// TIA Portal project "3motorfucnblock" (V20)

(* hardware
DEVICE "S7-1200 station_1"  S7-1200 Station
   slot 0: "Rack_0"  S7-1200 Rack  Rack  V1.0
   slot 1: "PLC_1"  CPU 1214C DC/DC/Rly  6ES7 214-1HG40-0XB0  V4.7
*)

// ===== PLC "PLC_1"  CPU 1214C DC/DC/Rly =====

VAR_GLOBAL   // PLC tag table "Default tag table"
   "Start but 1" AT %I0.0 : Bool;
   "Start but 2" AT %I0.1 : Bool;
   "Start but 3" AT %I0.2 : Bool;
   "Stop but 1" AT %I0.3 : Bool;
   "Stop but 2" AT %I0.4 : Bool;
   "Stop but 3" AT %I0.5 : Bool;
   "Reset but 1" AT %I0.6 : Bool;
   "Reset but 2" AT %I0.7 : Bool;
   "Reset but 3" AT %I1.0 : Bool;
   "Motor 1 çalış" AT %Q0.0 : Bool;
   "Motor 2 çalış" AT %Q0.1 : Bool;
   "Motor 3 çalış" AT %Q0.2 : Bool;
END_VAR

DATA_BLOCK "çalışma zamanları"   // DB1
{ S7_Optimized_Access := 'TRUE' }
VERSION : 0.1
   VAR
      "Motor 1 zaman" : Time := T#5s;
      "Motor 2 zaman" : Time := T#10s;
      "Motor 3 zaman" : Time := T#15s;
   END_VAR
BEGIN
END_DATA_BLOCK

DATA_BLOCK "çalışma sayıları"   // DB2
{ S7_Optimized_Access := 'TRUE' }
VERSION : 0.1
   VAR
      "Motor 1 sayı" : Int := 2;
      "Motor 2 sayı" : Int := 3;
      "Motor 3 sayı" : Int := 4;
   END_VAR
BEGIN
END_DATA_BLOCK

DATA_BLOCK "motor1"   // DB3
{ S7_Optimized_Access := 'TRUE' }
VERSION : 0.1
// stored: InstanceOfName Motorlar
"Motorlar"
BEGIN
END_DATA_BLOCK

DATA_BLOCK "motor2"   // DB4
{ S7_Optimized_Access := 'TRUE' }
VERSION : 0.1
// stored: InstanceOfName Motorlar
"Motorlar"
BEGIN
END_DATA_BLOCK

DATA_BLOCK "motor3"   // DB5
{ S7_Optimized_Access := 'TRUE' }
VERSION : 0.1
// stored: InstanceOfName Motorlar
"Motorlar"
BEGIN
END_DATA_BLOCK

FUNCTION_BLOCK "Motorlar"   // FB1, LAD
{ S7_Optimized_Access := 'TRUE' }
VERSION : 0.1
   VAR_INPUT
      Başlat : Bool;
      Durdur : Bool;
      Resetle : Bool;
      "Çalışma zamanı" : Time;
      "Çalışma sayısı" : Int;
   END_VAR
   VAR_OUTPUT
      "Motor çıkışı" : Bool;
   END_VAR
   VAR
      "Motor hafıza" : Bool;
      timer1 : TON_TIME;
      "Kenar darbesi" : Bool;
      "sayma sonucu" : Int;
      "Yeterli çalışma" : Bool;
   END_VAR
   VAR_TEMP   // added for the SCL form of the ladder/FBD networks
      _w1 : Bool;
   END_VAR
BEGIN

REGION Network 1
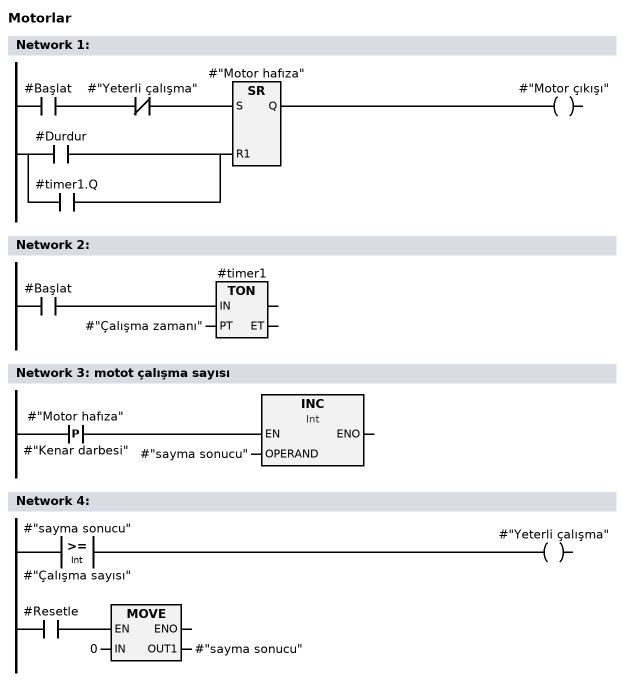
   RUNG wire#powerrail
      Contact( #Başlat )
      I_Contact( #"Yeterli çalışma" )
      S_SR(operand := #"Motor hafıza", r1 := wire#w1)
      Coil( #"Motor çıkışı" )
   END_RUNG
   RUNG wire#powerrail
      Contact( #Durdur )
   END_RUNG wire#w1
   RUNG wire#powerrail
      Contact( #timer1.Q )
   END_RUNG wire#w1
   // the same network as SCL:
   IF #Başlat AND NOT #"Yeterli çalışma" THEN
       #"Motor hafıza" := TRUE;   // SR flip-flop
   END_IF;
   IF #Durdur OR #timer1.Q THEN #"Motor hafıza" := FALSE; END_IF;
   #"Motor çıkışı" := #"Motor hafıza";
END_REGION

REGION Network 2
   #timer1(IN := #Başlat, PT := #"Çalışma zamanı");   // TON
END_REGION

REGION Network 3: motot çalışma sayısı
   RUNG wire#powerrail
      P_Contact(operand := #"Motor hafıza", bit := #"Kenar darbesi")
      { S7_Templates := "DestType := Int" } Inc( #"sayma sonucu" )
   END_RUNG
   // the same network as SCL:
   #_w1 := #"Motor hafıza" AND NOT #"Kenar darbesi";   // rising edge of #"Motor hafıza"
   #"Kenar darbesi" := #"Motor hafıza";
   IF #_w1 THEN #"sayma sonucu" := #"sayma sonucu" + 1; END_IF;
END_REGION

REGION Network 4
   RUNG wire#powerrail
      { S7_Templates := "SrcType := Int" } GE_Contact(in1 := #"sayma sonucu", in2 := #"Çalışma sayısı")
      Coil( #"Yeterli çalışma" )
   END_RUNG
   RUNG wire#powerrail
      Contact( #Resetle )
      Move(in := 0, out1 => #"sayma sonucu")
   END_RUNG
   // the same network as SCL:
   #"Yeterli çalışma" := #"sayma sonucu" >= #"Çalışma sayısı";
   IF #Resetle THEN #"sayma sonucu" := 0; END_IF;
END_REGION
END_FUNCTION_BLOCK

ORGANIZATION_BLOCK "Main"   // OB1, LAD, ProgramCycle
TITLE = "Main Program Sweep (Cycle)"
{ S7_Optimized_Access := 'TRUE' }
VERSION : 0.1
   VAR_INPUT
      Initial_Call : Bool;   // Initial call of this OB
      Remanence : Bool;   // =True, if remanent data are available
   END_VAR
BEGIN

REGION Network 1: Motor 1 çalışma programı
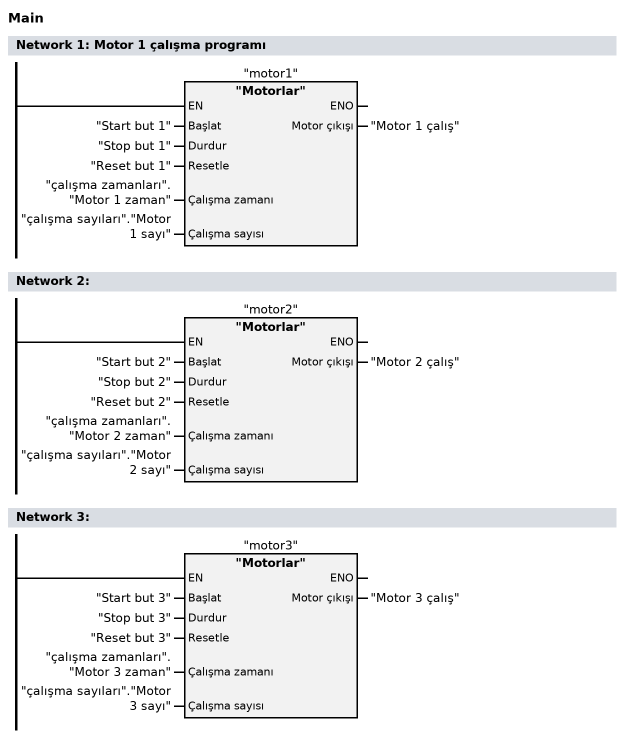
   RUNG wire#powerrail
      "motor1"(Başlat := "Start but 1", Durdur := "Stop but 1", Resetle := "Reset but 1", "Çalışma zamanı" := "çalışma zamanları"."Motor 1 zaman", "Çalışma sayısı" := "çalışma sayıları"."Motor 1 sayı", "Motor çıkışı" => "Motor 1 çalış")
   END_RUNG
   // the same network as SCL:
   "motor1"(Başlat := "Start but 1",   // "Motorlar"
            Durdur := "Stop but 1",
            Resetle := "Reset but 1",
            "Çalışma zamanı" := "çalışma zamanları"."Motor 1 zaman",
            "Çalışma sayısı" := "çalışma sayıları"."Motor 1 sayı",
            "Motor çıkışı" => "Motor 1 çalış");
END_REGION

REGION Network 2
   RUNG wire#powerrail
      "motor2"(Başlat := "Start but 2", Durdur := "Stop but 2", Resetle := "Reset but 2", "Çalışma zamanı" := "çalışma zamanları"."Motor 2 zaman", "Çalışma sayısı" := "çalışma sayıları"."Motor 2 sayı", "Motor çıkışı" => "Motor 2 çalış")
   END_RUNG
   // the same network as SCL:
   "motor2"(Başlat := "Start but 2",   // "Motorlar"
            Durdur := "Stop but 2",
            Resetle := "Reset but 2",
            "Çalışma zamanı" := "çalışma zamanları"."Motor 2 zaman",
            "Çalışma sayısı" := "çalışma sayıları"."Motor 2 sayı",
            "Motor çıkışı" => "Motor 2 çalış");
END_REGION

REGION Network 3
   RUNG wire#powerrail
      "motor3"(Başlat := "Start but 3", Durdur := "Stop but 3", Resetle := "Reset but 3", "Çalışma zamanı" := "çalışma zamanları"."Motor 3 zaman", "Çalışma sayısı" := "çalışma sayıları"."Motor 3 sayı", "Motor çıkışı" => "Motor 3 çalış")
   END_RUNG
   // the same network as SCL:
   "motor3"(Başlat := "Start but 3",   // "Motorlar"
            Durdur := "Stop but 3",
            Resetle := "Reset but 3",
            "Çalışma zamanı" := "çalışma zamanları"."Motor 3 zaman",
            "Çalışma sayısı" := "çalışma sayıları"."Motor 3 sayı",
            "Motor çıkışı" => "Motor 3 çalış");
END_REGION
END_ORGANIZATION_BLOCK